% RSLogix 500 project send_data.RSS, saved by version 8.30.00.15 %
PROJECT "UNTITLED"    % processor: Bul.1763 MicroLogix 1100 Series A %

PROGRAM FILES
  LAD 2 "MAIN"  5 rungs
  LAD 3 "SEND_DATA"  1 rungs

DATA FILES
  O0 OUTPUT  4 elements
  I1 INPUT  6 elements
  S2 STATUS  66 elements
  B3 BINARY  1 elements
  T4 TIMER  2 elements
  C5 COUNTER  1 elements
  R6 CONTROL  1 elements
  N7 INTEGER  4 elements
  F8 FLOAT  1 elements

LADDER 2 "MAIN"
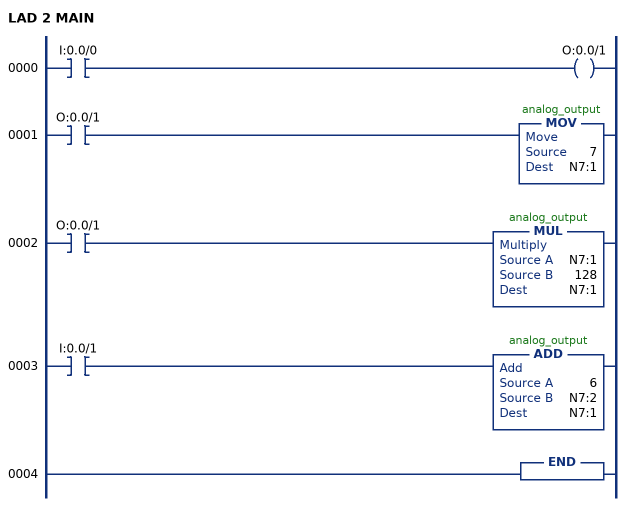
% Rung: 0 %
SOR XIC I:0.0/0 OTE O:0.0/1 EOR
% Rung: 1 %
SOR XIC O:0.0/1 MOV 7 N7:1 EOR
%   N7:1  "analog_output" %
% Rung: 2 %
SOR XIC O:0.0/1 MUL N7:1 128 N7:1 EOR
%   N7:1  "analog_output" %
% Rung: 3 %
SOR XIC I:0.0/1 ADD 6 N7:2 N7:1 EOR
%   N7:1  "analog_output" %
% Rung: 4 %
SOR END EOR

OTHER DOCUMENTED ADDRESSES
  5_  
